TYPE UDT_BinList :
STRUCT
	Bin: ARRAY[0..255] OF  UDT_Bin;
	arWorkPos: ARRAY[1..40] OF LREAL;
	arInRang: ARRAY[1..40] OF BOOL;
	Reset: BOOL;
END_STRUCT
END_TYPE

(* stored: Version 1.1.0.1, ProductVersion 3.1.4022.16
   DUT UDT_BinList: Id {34d64548-72bb-4d23-9424-0d23fe43e1fd} *)
